{attribute 'GeneratedUsingTerminal: KL2641'}
{attribute addProperty BoxType "KL2641"}
{attribute addProperty Description ""}
{attribute addProperty Physics ""}
{attribute addProperty Id "Channel_1AT %Q*Channel_2589C8DC0"}
{attribute addProperty CRC "2223485445"}
{attribute addProperty Size "0"}
TYPE KL2641_8487B205 :
STRUCT
	{attribute addProperty Name "Channel_1"}
	Channel_1 : Channel_2589C8DC;
END_STRUCT
END_TYPE

(* stored: Version 1.2.0.0, ProductVersion 3.1.4024.11
   DUT KL2641_8487B205: Id {2e789d50-88cc-4de5-8140-152c59f201aa} *)
